PROGRAM Main_Vacuum
VAR
END_VAR

IF NOT Vacuum_Buffer_Data.Vacuumed THEN
	Vacuum_Buffer_Data();
END_IF

IF NOT Vacuum_Buffer_IMU.Vacuumed THEN
	Vacuum_Buffer_IMU();
END_IF

IF NOT Vacuum_Buffer_IMU_2.Vacuumed THEN
	Vacuum_Buffer_IMU_2();
END_IF

IF NOT Vacuum_Data.Vacuumed THEN
	Vacuum_Data();
END_IF

IF NOT Vacuum_IMU.Vacuumed THEN
	Vacuum_IMU();
END_IF

END_PROGRAM

(* stored: Version 1.1.0.1, ProductVersion 3.1.4024.6
   POU Main_Vacuum: Id {08fdd8cd-369e-485f-a484-135431d0cebb}, SpecialFunc None *)
